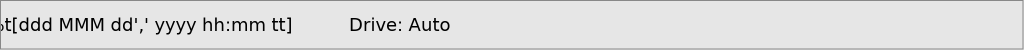
VISUALIZATION StatusBar  // 1024x50
    Textfield (-35,0 350x50), "%t[ddd MMM dd',' yyyy hh:mm tt]", text variable: HARV.TimeTracker.TimeStampStruct
    Textfield (325,0 150x50), "Drive: Auto"
END_VISUALIZATION

(* stored: Version 1.1.0.1, ProductVersion 3.1.4024.12
   Visu StatusBar: Id {fd191f35-689c-4162-8c7a-1034e5e00885} *)
